// Mitsubishi GX Works2 project: 6   PLC: FX3U/FX3UC

// task Task_01 (event TRUE, interval 0, priority 31): POU_01

PROGRAM POU_01
VAR
  cnt : INT;
  ii : INT;
  wstep : INT;
  rt : R_TRIG;
  rt2 : R_TRIG;
END_VAR
rt(_CLK := M0);
rt2(_CLK := M1);

IF rt.Q THEN
	cnt := cnt + 1;
	cnt := cnt MOD 4;
END_IF;

IF M1 OR M8002 THEN
	cnt := 0;
END_IF;

FOR ii := 1 TO 4 BY 1 DO
	Z0 := ii;
	Y0Z0 := FALSE;
END_FOR;

FOR ii := 1 TO cnt BY 1 DO
	Z1 := ii;
	Y0Z1 := TRUE;
END_FOR;
END_PROGRAM
